TYPE TrackInfo :
STRUCT
	TrackId 				: OTCID;	// hardware id of mover's track read back from MC_ReadTrackPositions
	PartId 					: OTCID;	// hardware id of mover's part read back from MC_ReadTrackPositions
	TrackPosition 			: LREAL;	// track position read back from MC_ReadTrackPositions
	PartPosition			: LREAL;	// part position read back from MC_ReadTrackPositions
END_STRUCT
END_TYPE

(* stored: Version 1.1.0.1, ProductVersion 3.1.4026.8
   DUT TrackInfo: Id {e1df8d7d-bb5e-01fd-14ad-401c12b84a9f} *)
